% RSLogix 500 project P1_ABIOLA_A_TESTING V9_BAK270.RSS, saved by version 8.30.00.16 %
PROJECT "UNTITLED"    % processor: Bul.1763 MicroLogix 1100 Series B %

PROGRAM FILES
  LAD 2   4 rungs
  LAD 3 "INPUT DVS"  3 rungs  % This contains all input addresses linked to bits %
  LAD 4 "OUTPUT DVS"  3 rungs  % This contains addresses to output devices  %
  LAD 5 "PRO LOGIC"  4 rungs  % This contains how the process is implemented %

DATA FILES
  O0 OUTPUT  4 elements
  I1 INPUT  6 elements
  S2 STATUS  66 elements
  B3 BINARY  1 elements
  T4 TIMER  1 elements
  C5 COUNTER  1 elements
  R6 CONTROL  1 elements
  N7 INTEGER  2 elements
  F8 FLOAT  1 elements

LADDER 2
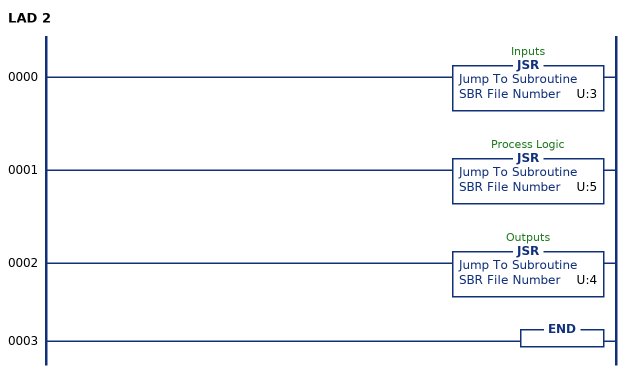
% Rung: 0 %
SOR JSR U:3 EOR
%   U:3  "Inputs" %
% Rung: 1 %
SOR JSR U:5 EOR
%   U:5  "Process Logic" %
% Rung: 2 %
SOR JSR U:4 EOR
%   U:4  "Outputs" %
% Rung: 3 %
SOR END EOR

LADDER 3 "INPUT DVS"    % This contains all input addresses linked to bits %
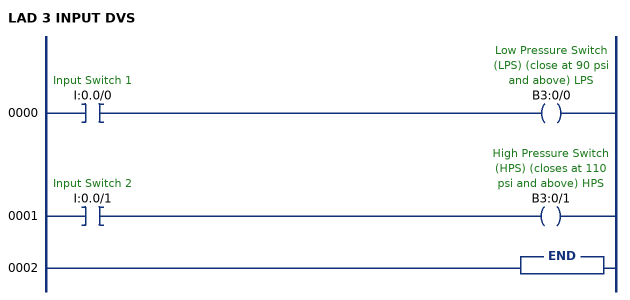
% Rung: 0 %
SOR XIC I:0.0/0 OTE B3:0/0 EOR
%   I:0.0/0  "Input Switch 1" %
%   B3:0/0  LPS  "Low Pressure Switch (LPS) (close at 90 psi and above)" %
% Rung: 1 %
SOR XIC I:0.0/1 OTE B3:0/1 EOR
%   I:0.0/1  "Input Switch 2" %
%   B3:0/1  HPS  "High Pressure Switch (HPS) (closes at 110 psi and above)" %
% Rung: 2 %
SOR END EOR

LADDER 4 "OUTPUT DVS"    % This contains addresses to output devices  %
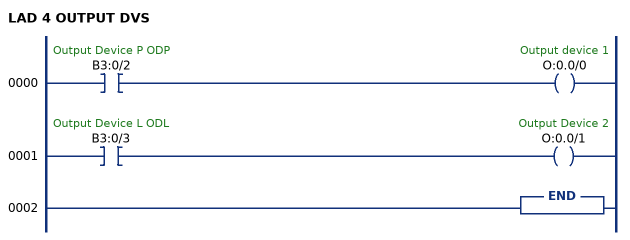
% Rung: 0 %
SOR XIC B3:0/2 OTE O:0.0/0 EOR
%   B3:0/2  ODP  "Output Device P" %
%   O:0.0/0  "Output device 1" %
% Rung: 1 %
SOR XIC B3:0/3 OTE O:0.0/1 EOR
%   B3:0/3  ODL  "Output Device L" %
%   O:0.0/1  "Output Device 2" %
% Rung: 2 %
SOR END EOR

LADDER 5 "PRO LOGIC"    % This contains how the process is implemented %
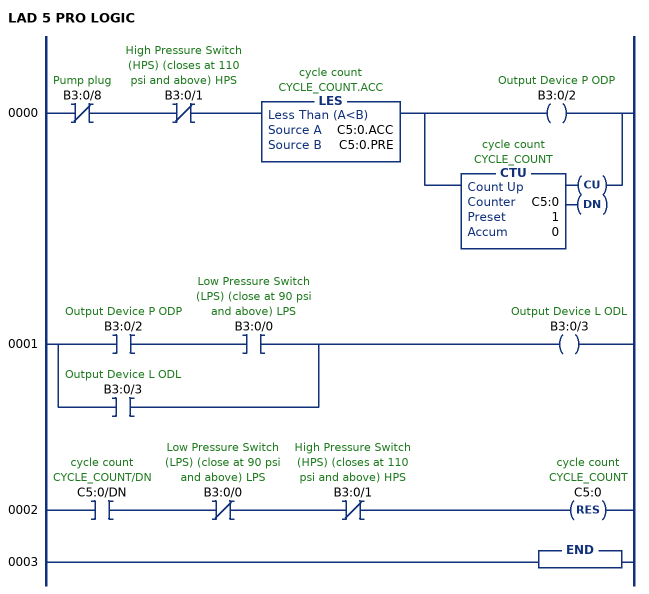
% Rung: 0 %
SOR XIO B3:0/8 XIO B3:0/1 LES C5:0.ACC C5:0.PRE BST OTE B3:0/2 NXB CTU C5:0 1 0 BND EOR
%   B3:0/8  "Pump plug" %
%   B3:0/1  HPS  "High Pressure Switch (HPS) (closes at 110 psi and above)" %
%   C5:0  CYCLE_COUNT  "cycle count" %
%   B3:0/2  ODP  "Output Device P" %
% Rung: 1 %
SOR BST XIC B3:0/2 XIC B3:0/0 NXB XIC B3:0/3 BND OTE B3:0/3 EOR
%   B3:0/2  ODP  "Output Device P" %
%   B3:0/0  LPS  "Low Pressure Switch (LPS) (close at 90 psi and above)" %
%   B3:0/3  ODL  "Output Device L" %
% Rung: 2 %  % edit flag set %
SOR XIC C5:0/DN XIO B3:0/0 XIO B3:0/1 RES C5:0 EOR
%   C5:0  CYCLE_COUNT  "cycle count" %
%   B3:0/0  LPS  "Low Pressure Switch (LPS) (close at 90 psi and above)" %
%   B3:0/1  HPS  "High Pressure Switch (HPS) (closes at 110 psi and above)" %
% Rung: 3 %
SOR END EOR

OTHER DOCUMENTED ADDRESSES
  B3:0/4  "One shot"
  B3:0/5  "One shot 2"
  B3:0/6  "One shot 3"
  B3:0/7  "One shot 4"
  N7:0  LPS_ACTIVATED  "LPS_activated (if psi = 90)"
  N7:1  HPS_ACTIVATED  "HPS_activated"
  T4:0  TIMER  "Timer EN - Energized once true DN- Energized after preset value"
  T4:0/DN  DN_TIMER
  T4:0/EN  EN_TIMER  "De-energized when psi > 90"

DATA TABLE (non-zero values as saved)
DATA T4
% .PRE .ACC %
% T4:0 % 1 0
DATA C5
% .PRE .ACC %
% C5:0 % 1 0
